Yaskawa INFORM job: CVAR_EXAMPLE.JBI

/JOB
//NAME INFORM_SYNTAX_4
//POS
///NPOS 3,0,0,0,0,0
///TOOL 0
///POSTYPE PULSE
///PULSE
C00000=0,0,0,0,0,0,0
C00001=-47130,2431,-2253,2953,1210,-10822,-112862
C00002=0,0,0,0,0,0,0
//INST
///DATE 2011/12/21 00:50
///ATTR SC,RW
///GROUP1 RB1
NOP
IFTHEN I000=-32768
ELSEIF IN#(1)=ON
ENDIF
MOVJ C00000 VJ=0.78
MOVJ C00001 VJ=0.78
MOVJ C00002 VJ=0.78
END
